PROGRAM AutoStartCtrl
VAR

	PV: TIME;
	tUldPos1BasketMemoryReset: TON;
	tUldPos2BasketMemoryReset: TON;
	tUldPos3BasketMemoryReset: TON;
	tUldPos4BasketMemoryReset: TON;
	tUldPos5BasketMemoryReset: TON;

	tLdPos1BasketMemoryReset: TON;
	tLdPos2BasketMemoryReset: TON;
	tLdPos3BasketMemoryReset: TON;
	tLdPos4BasketMemoryReset: TON;
	tLdPos5BasketMemoryReset: TON;

	tUld1BasketMemoryReset: TON;
	tUld2BasketMemoryReset: TON;
	tUld1BasketMemoryWriteIn: TON;
	ULDTimer: TON;
	ULDSingleBasketReachedTimer: TON;

	tLd1BasketMemoryIndexReset: TON;

	ULDBuzzerOffHeaterTimer: TON;

END_VAR
VAR // added by the converter: edge detectors and wires of the graphical bodies
    _w1, _w2, _w3 : INT;
END_VAR

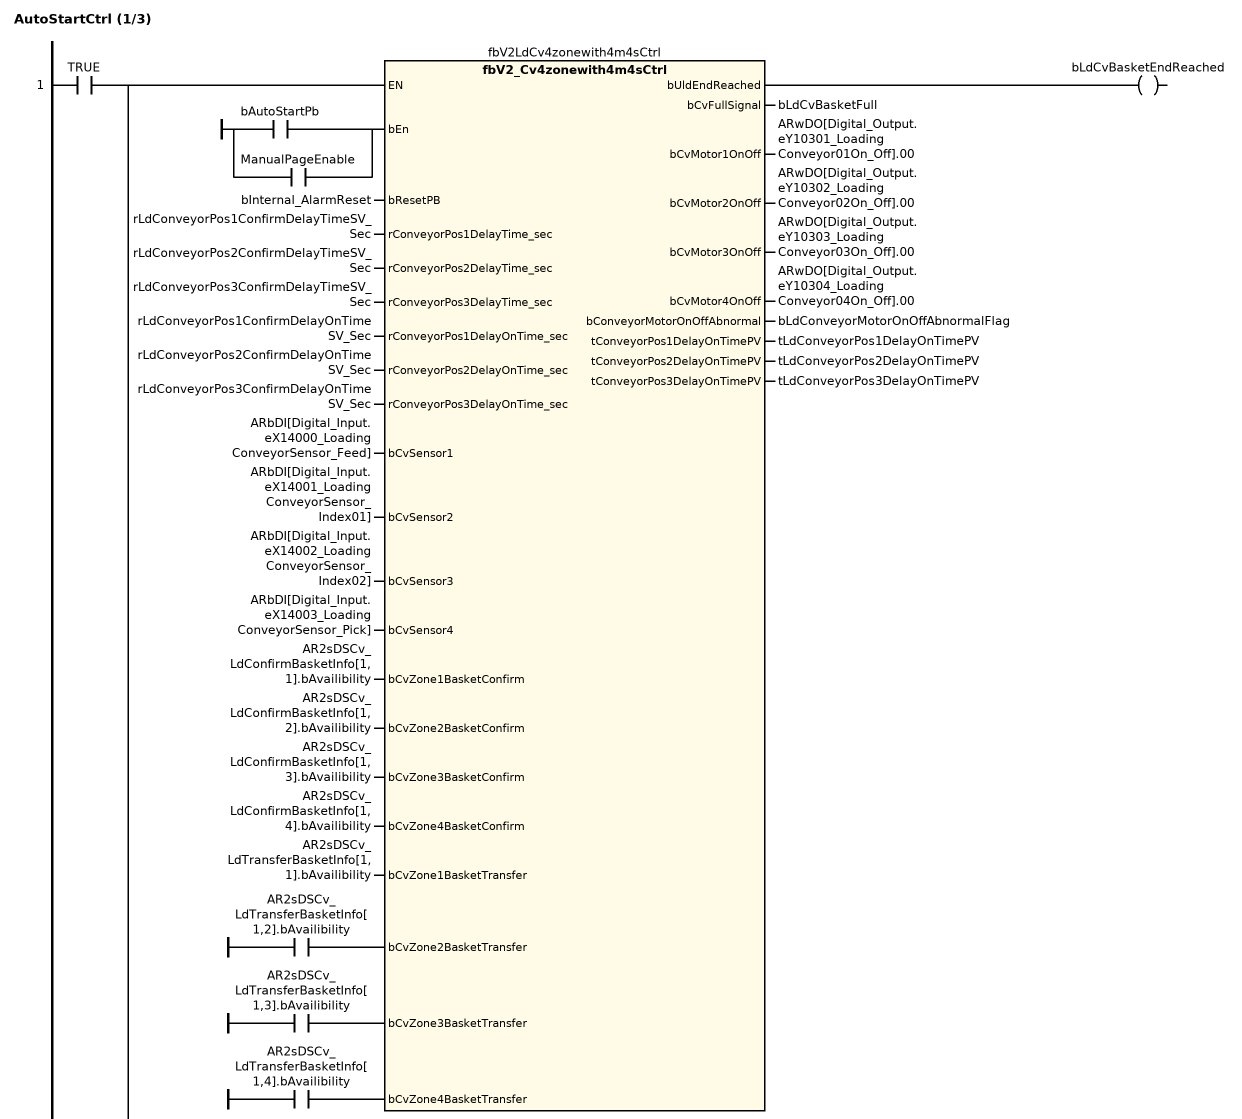
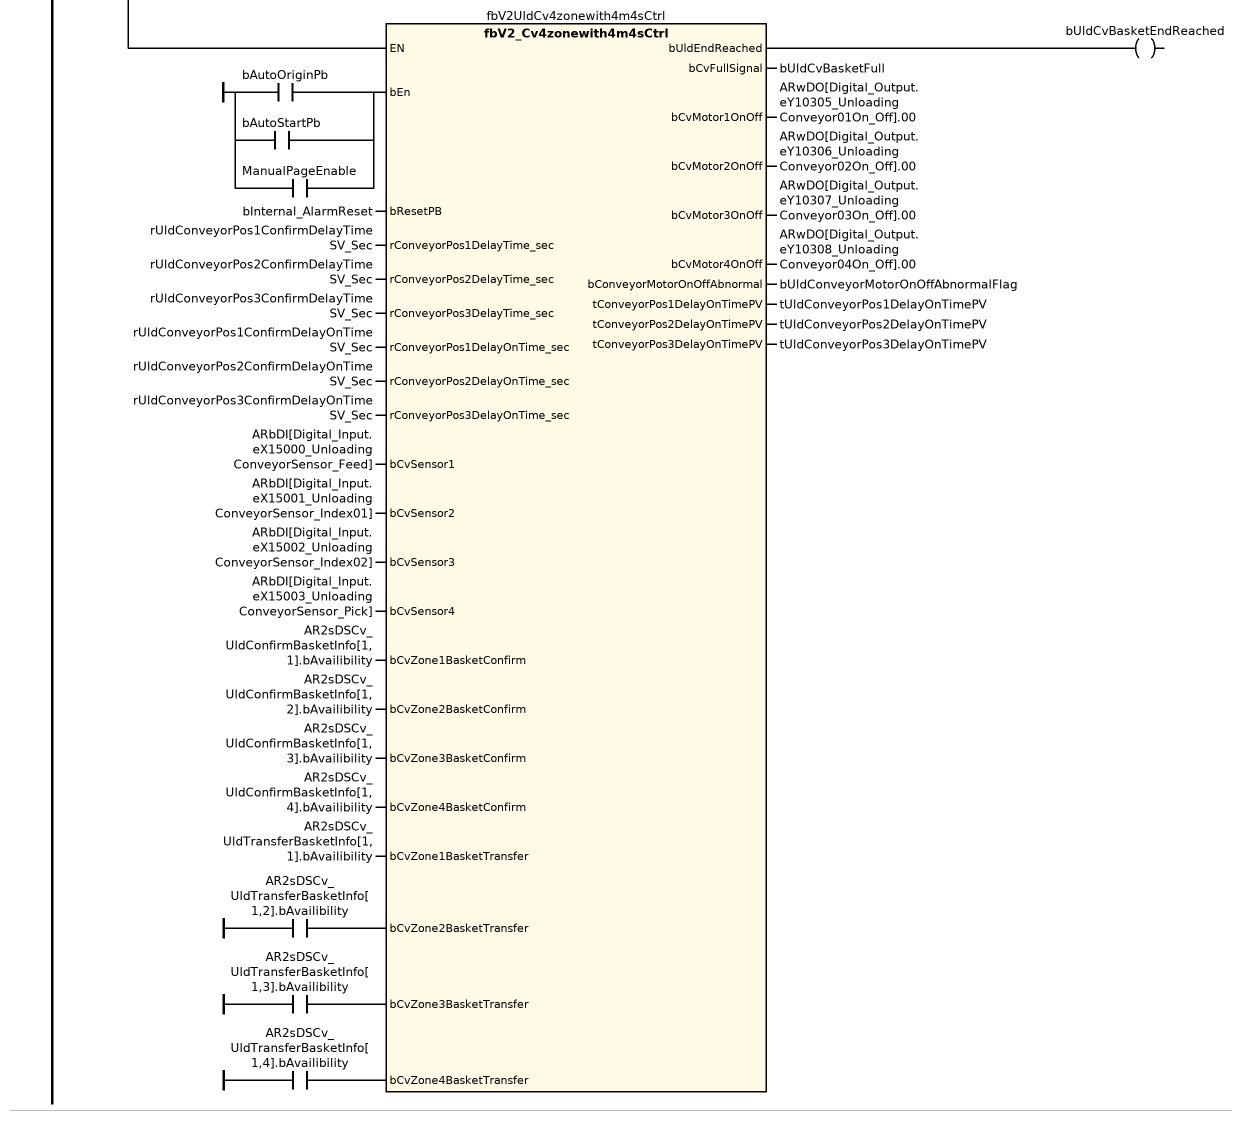
// NETWORK 1
fbV2LdCv4zonewith4m4sCtrl(
    bEn := bAutoStartPb OR ManualPageEnable,
    bResetPB := bInternal_AlarmReset,
    rConveyorPos1DelayTime_sec := rLdConveyorPos1ConfirmDelayTimeSV_Sec,
    rConveyorPos2DelayTime_sec := rLdConveyorPos2ConfirmDelayTimeSV_Sec,
    rConveyorPos3DelayTime_sec := rLdConveyorPos3ConfirmDelayTimeSV_Sec,
    rConveyorPos1DelayOnTime_sec := rLdConveyorPos1ConfirmDelayOnTimeSV_Sec,
    rConveyorPos2DelayOnTime_sec := rLdConveyorPos2ConfirmDelayOnTimeSV_Sec,
    rConveyorPos3DelayOnTime_sec := rLdConveyorPos3ConfirmDelayOnTimeSV_Sec,
    bCvSensor1 := ARbDI[Digital_Input.eX14000_LoadingConveyorSensor_Feed],
    bCvSensor2 := ARbDI[Digital_Input.eX14001_LoadingConveyorSensor_Index01],
    bCvSensor3 := ARbDI[Digital_Input.eX14002_LoadingConveyorSensor_Index02],
    bCvSensor4 := ARbDI[Digital_Input.eX14003_LoadingConveyorSensor_Pick],
    bCvZone1BasketConfirm := AR2sDSCv_LdConfirmBasketInfo[1,1].bAvailibility,
    bCvZone2BasketConfirm := AR2sDSCv_LdConfirmBasketInfo[1,2].bAvailibility,
    bCvZone3BasketConfirm := AR2sDSCv_LdConfirmBasketInfo[1,3].bAvailibility,
    bCvZone4BasketConfirm := AR2sDSCv_LdConfirmBasketInfo[1,4].bAvailibility,
    bCvZone1BasketTransfer := AR2sDSCv_LdTransferBasketInfo[1,1].bAvailibility,
    bCvZone2BasketTransfer := AR2sDSCv_LdTransferBasketInfo[1,2].bAvailibility,
    bCvZone3BasketTransfer := AR2sDSCv_LdTransferBasketInfo[1,3].bAvailibility,
    bCvZone4BasketTransfer := AR2sDSCv_LdTransferBasketInfo[1,4].bAvailibility,
    bCvFullSignal => bLdCvBasketFull,
    bCvMotor1OnOff => ARwDO[Digital_Output.eY10301_LoadingConveyor01On_Off].00,
    bCvMotor2OnOff => ARwDO[Digital_Output.eY10302_LoadingConveyor02On_Off].00,
    bCvMotor3OnOff => ARwDO[Digital_Output.eY10303_LoadingConveyor03On_Off].00,
    bCvMotor4OnOff => ARwDO[Digital_Output.eY10304_LoadingConveyor04On_Off].00,
    bConveyorMotorOnOffAbnormal => bLdConveyorMotorOnOffAbnormalFlag,
    tConveyorPos1DelayOnTimePV => tLdConveyorPos1DelayOnTimePV,
    tConveyorPos2DelayOnTimePV => tLdConveyorPos2DelayOnTimePV,
    tConveyorPos3DelayOnTimePV => tLdConveyorPos3DelayOnTimePV); // fbV2_Cv4zonewith4m4sCtrl
bLdCvBasketEndReached := fbV2LdCv4zonewith4m4sCtrl.bUldEndReached;
fbV2UldCv4zonewith4m4sCtrl(
    bEn := bAutoOriginPb OR bAutoStartPb OR ManualPageEnable,
    bResetPB := bInternal_AlarmReset,
    rConveyorPos1DelayTime_sec := rUldConveyorPos1ConfirmDelayTimeSV_Sec,
    rConveyorPos2DelayTime_sec := rUldConveyorPos2ConfirmDelayTimeSV_Sec,
    rConveyorPos3DelayTime_sec := rUldConveyorPos3ConfirmDelayTimeSV_Sec,
    rConveyorPos1DelayOnTime_sec := rUldConveyorPos1ConfirmDelayOnTimeSV_Sec,
    rConveyorPos2DelayOnTime_sec := rUldConveyorPos2ConfirmDelayOnTimeSV_Sec,
    rConveyorPos3DelayOnTime_sec := rUldConveyorPos3ConfirmDelayOnTimeSV_Sec,
    bCvSensor1 := ARbDI[Digital_Input.eX15000_UnloadingConveyorSensor_Feed],
    bCvSensor2 := ARbDI[Digital_Input.eX15001_UnloadingConveyorSensor_Index01],
    bCvSensor3 := ARbDI[Digital_Input.eX15002_UnloadingConveyorSensor_Index02],
    bCvSensor4 := ARbDI[Digital_Input.eX15003_UnloadingConveyorSensor_Pick],
    bCvZone1BasketConfirm := AR2sDSCv_UldConfirmBasketInfo[1,1].bAvailibility,
    bCvZone2BasketConfirm := AR2sDSCv_UldConfirmBasketInfo[1,2].bAvailibility,
    bCvZone3BasketConfirm := AR2sDSCv_UldConfirmBasketInfo[1,3].bAvailibility,
    bCvZone4BasketConfirm := AR2sDSCv_UldConfirmBasketInfo[1,4].bAvailibility,
    bCvZone1BasketTransfer := AR2sDSCv_UldTransferBasketInfo[1,1].bAvailibility,
    bCvZone2BasketTransfer := AR2sDSCv_UldTransferBasketInfo[1,2].bAvailibility,
    bCvZone3BasketTransfer := AR2sDSCv_UldTransferBasketInfo[1,3].bAvailibility,
    bCvZone4BasketTransfer := AR2sDSCv_UldTransferBasketInfo[1,4].bAvailibility,
    bCvFullSignal => bUldCvBasketFull,
    bCvMotor1OnOff => ARwDO[Digital_Output.eY10305_UnloadingConveyor01On_Off].00,
    bCvMotor2OnOff => ARwDO[Digital_Output.eY10306_UnloadingConveyor02On_Off].00,
    bCvMotor3OnOff => ARwDO[Digital_Output.eY10307_UnloadingConveyor03On_Off].00,
    bCvMotor4OnOff => ARwDO[Digital_Output.eY10308_UnloadingConveyor04On_Off].00,
    bConveyorMotorOnOffAbnormal => bUldConveyorMotorOnOffAbnormalFlag,
    tConveyorPos1DelayOnTimePV => tUldConveyorPos1DelayOnTimePV,
    tConveyorPos2DelayOnTimePV => tUldConveyorPos2DelayOnTimePV,
    tConveyorPos3DelayOnTimePV => tUldConveyorPos3DelayOnTimePV); // fbV2_Cv4zonewith4m4sCtrl
bUldCvBasketEndReached := fbV2UldCv4zonewith4m4sCtrl.bUldEndReached;

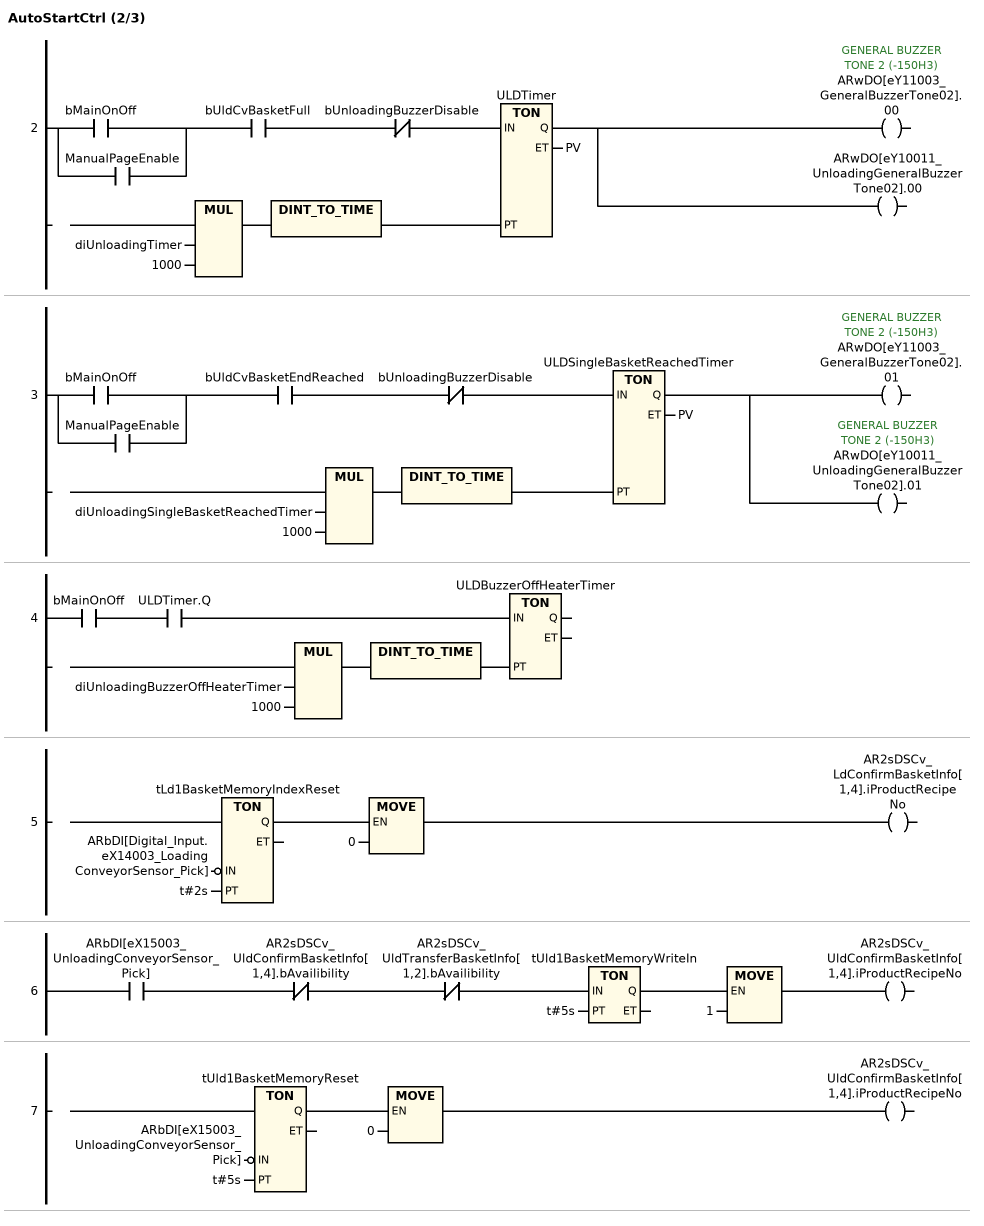
// NETWORK 2
//   ARwDO[eY11003_GeneralBuzzerTone02].00: GENERAL BUZZER TONE 2 (-150H3)
ULDTimer(
    IN := (bMainOnOff OR ManualPageEnable) AND bUldCvBasketFull AND NOT bUnloadingBuzzerDisable,
    PT := DINT_TO_TIME(diUnloadingTimer * 1000),
    ET => PV); // TON
ARwDO[eY11003_GeneralBuzzerTone02].00 := ULDTimer.Q;
ARwDO[eY10011_UnloadingGeneralBuzzerTone02].00 := ULDTimer.Q;

// NETWORK 3
//   ARwDO[eY11003_GeneralBuzzerTone02].01: GENERAL BUZZER TONE 2 (-150H3)
//   ARwDO[eY10011_UnloadingGeneralBuzzerTone02].01: GENERAL BUZZER TONE 2 (-150H3)
ULDSingleBasketReachedTimer(
    IN := (bMainOnOff OR ManualPageEnable) AND bUldCvBasketEndReached AND NOT bUnloadingBuzzerDisable,
    PT := DINT_TO_TIME(diUnloadingSingleBasketReachedTimer * 1000),
    ET => PV); // TON
ARwDO[eY11003_GeneralBuzzerTone02].01 := ULDSingleBasketReachedTimer.Q;
ARwDO[eY10011_UnloadingGeneralBuzzerTone02].01 := ULDSingleBasketReachedTimer.Q;

// NETWORK 4
ULDBuzzerOffHeaterTimer(IN := bMainOnOff AND ULDTimer.Q, PT := DINT_TO_TIME(diUnloadingBuzzerOffHeaterTimer * 1000)); // TON

// NETWORK 5
tLd1BasketMemoryIndexReset(IN := NOT ARbDI[Digital_Input.eX14003_LoadingConveyorSensor_Pick], PT := t#2s); // TON
IF tLd1BasketMemoryIndexReset.Q THEN _w1 := 0; END_IF
AR2sDSCv_LdConfirmBasketInfo[1,4].iProductRecipeNo := _w1;

// NETWORK 6
tUld1BasketMemoryWriteIn(IN := ARbDI[eX15003_UnloadingConveyorSensor_Pick] AND NOT AR2sDSCv_UldConfirmBasketInfo[1,4].bAvailibility AND NOT AR2sDSCv_UldTransferBasketInfo[1,2].bAvailibility, PT := t#5s); // TON
IF tUld1BasketMemoryWriteIn.Q THEN _w2 := 1; END_IF
AR2sDSCv_UldConfirmBasketInfo[1,4].iProductRecipeNo := _w2;

// NETWORK 7
tUld1BasketMemoryReset(IN := NOT ARbDI[eX15003_UnloadingConveyorSensor_Pick], PT := t#5s); // TON
IF tUld1BasketMemoryReset.Q THEN _w3 := 0; END_IF
AR2sDSCv_UldConfirmBasketInfo[1,4].iProductRecipeNo := _w3;

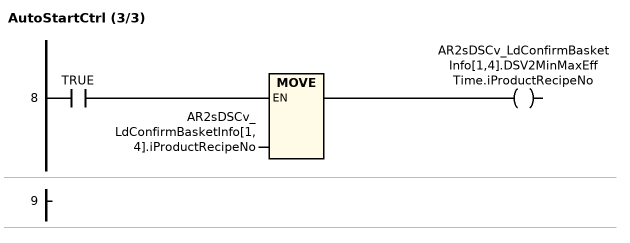
// NETWORK 8
AR2sDSCv_LdConfirmBasketInfo[1,4].DSV2MinMaxEffTime.iProductRecipeNo := AR2sDSCv_LdConfirmBasketInfo[1,4].iProductRecipeNo;

// NETWORK 9

ACTION ACT:
AR2sDSCv_UldTransferBasketInfo[1,4].iProductRecipeNo:=0;
AR2sDSCv_LdTransferBasketInfo[1,4].iProductRecipeNo:=0;
END_ACTION

END_PROGRAM

(* stored: Version 1.1.0.1, ProductVersion 3.1.4024.12
   POU AutoStartCtrl: Id {b80143e4-d88b-46b3-aea3-f927ab7282b9}, SpecialFunc None
   Action ACT: Id {40ee3928-b053-408f-86b1-4567415a35f8} *)
